(* PLC project Tub_1, Beckhoff Automation GmbH TwinCAT PLC Control 3.5.13.21 *)
(* stored: creationDateTime 2022-03-23T14:57:37.7517656, modificationDateTime 2022-03-23T14:57:37.7547638 *)

(* global variable list GVL *)
{attribute 'qualified_only'}
VAR_GLOBAL
	
	mb_Input_Coils			: ARRAY [0..255] OF BOOL;
	mb_Output_Coils			: ARRAY [0..255] OF BOOL;
	mb_Input_Registers		: ARRAY [0..255] OF WORD;
	mb_Output_Registers		: ARRAY [0..255] OF WORD;
	
END_VAR
